Fanuc TP program (LS listing): EOAT_OPEN.LS

/PROG  EOAT_OPEN	  Macro
/ATTR
OWNER		= MNEDITOR;
COMMENT		= "";
PROG_SIZE	= 209;
CREATE		= DATE 19-08-13  TIME 08:00:42;
MODIFIED	= DATE 19-08-13  TIME 08:01:02;
FILE_NAME	= ;
VERSION		= 0;
LINE_COUNT	= 2;
MEMORY_SIZE	= 589;
PROTECT		= READ_WRITE;
TCD:  STACK_SIZE	= 0,
      TASK_PRIORITY	= 50,
      TIME_SLICE	= 0,
      BUSY_LAMP_OFF	= 0,
      ABORT_REQUEST	= 0,
      PAUSE_REQUEST	= 0;
DEFAULT_GROUP	= *,*,*,*,*;
CONTROL_CODE	= 00000000 00000000;
/APPL

AUTO_SINGULARITY_HEADER;
  ENABLE_SINGULARITY_AVOIDANCE   : FALSE;
/MN
   1:  CALL CLAMP_OPEN    ;
   2:  CALL GRIPPER_OPEN    ;
/POS
/END
